FUNCTION_BLOCK Section5Ctrl
  (* Standard: 61499-2 *)
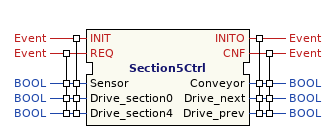
  EVENT_INPUT
    INIT WITH Sensor, Drive_section0, Drive_section4;
    REQ WITH Sensor, Drive_section0, Drive_section4;
  END_EVENT
  EVENT_OUTPUT
    INITO WITH Conveyor, Drive_next, Drive_prev;
    CNF WITH Conveyor, Drive_next, Drive_prev;
  END_EVENT
  VAR_INPUT
    Sensor : BOOL;
    Drive_section0 : BOOL;
    Drive_section4 : BOOL;
  END_VAR
  VAR_OUTPUT
    Conveyor : BOOL;
    Drive_next : BOOL;
    Drive_prev : BOOL;
  END_VAR
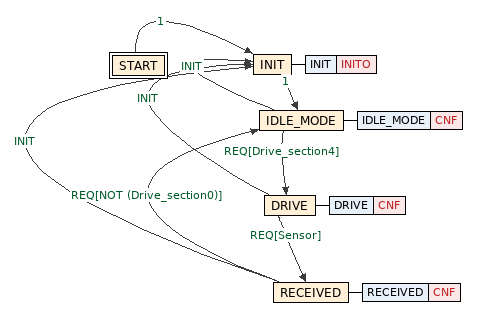
  EC_STATES
    START;
    INIT : INIT -> INITO;
    IDLE_MODE : IDLE_MODE -> CNF;
    DRIVE : DRIVE -> CNF;
    RECEIVED : RECEIVED -> CNF;
  END_STATES
  EC_TRANSITIONS
    START TO INIT := 1;
    INIT TO IDLE_MODE := 1;
    IDLE_MODE TO DRIVE := REQ[Drive_section4];
    DRIVE TO RECEIVED := REQ[Sensor];
    RECEIVED TO IDLE_MODE := REQ[NOT (Drive_section0)];
    IDLE_MODE TO INIT := INIT;
    DRIVE TO INIT := INIT;
    RECEIVED TO INIT := INIT;
  END_TRANSITIONS
  ALGORITHM INIT IN ST:
Conveyor := FALSE;&#10;Drive_prev := FALSE;&#10;Drive_next := FALSE;&#10;
  END_ALGORITHM
  ALGORITHM IDLE_MODE IN ST:
Conveyor := FALSE;&#10;Drive_prev := TRUE;&#10;Drive_next := FALSE;&#10;
  END_ALGORITHM
  ALGORITHM DRIVE IN ST:
Conveyor := TRUE;&#10;Drive_prev := TRUE;&#10;Drive_next := FALSE;&#10;
  END_ALGORITHM
  ALGORITHM RECEIVED IN ST:
Conveyor := TRUE;&#10;Drive_prev := FALSE;&#10;Drive_next := TRUE;&#10;
  END_ALGORITHM
END_FUNCTION_BLOCK
